Omron Sysmac Studio project Project-Backup-Onrom (Sysmac Studio 1.64.0.64008, StandardProject)

# Controller CLP: NX102-1020 version 1.33
Units and slaves: Unit 1 : NX-ID5442 (N1); Unit 2 : NX-OD5256 (N2); Unit 3 : NX-PF0730 (N3); Unit 5 : NX-SID800 (N5); Unit 6 : NX-SOD400 (N6)
Axis MC_Axis000, settings changed from default: AxisType=ServoType, UnitsConversion=EnumElement2, UnitsNumerator=8388608, UnitsDenominator=100, MaxVelocity=10000, MaxJogVelocity=8000, MaxAcceleration=50, MaxDeceleration=50, MaxPositiveTorqueLimit=050.0, MaxNegativeTorqueLimit=050.0, HomingMode=BackupAndProximitySignalOn, StartDirection=NegativeDirection, OriginInputDetectionDirection=NegativeDirection, HomingVelocity=100, HomingApproachVelocity=5, OriginCompensationValue=10, CompensationVelocity=5, ModuloMAXPosition=100, ModuloMINPosition=0, EncoderTypes=Abs
Task PrimaryTask (priority 4, period or condition 2000): Program0

VAR_GLOBAL
    PB1 : BOOL;  (* IHM; published *)
    O1 : BOOL;  (* at IOBus://unit#2/Output Bit 16 bits/Output Bit 01 *)
END_VAR
VAR_GLOBAL CONSTANT
    MC_Axis000 : _sAXIS_REF;  (* at MC://_MC_AX[0] *)
END_VAR
VAR_GLOBAL
    O2 : BOOL;  (* at IOBus://unit#2/Output Bit 16 bits/Output Bit 02 *)
    O3 : BOOL;  (* at IOBus://unit#2/Output Bit 16 bits/Output Bit 03 *)
    PBSET : BOOL;  (* IHM; published *)
    PBRESET : BOOL;  (* IHM; published *)
    PBMOMENT : BOOL;
    LPOUT02 : BOOL;
    LPOUT03 : BOOL;
    PBM_LIG : BOOL;  (* IHM; published *)
    PBM_DSL : BOOL;  (* IHM; published *)
    TEMPO_O2 : TIME;
    PV : DINT;
    SP : DINT;
    E001_Torque_actual_value : INT;  (* at ECAT://node#1/Torque actual value; published *)
    Torque_atual : INT;  (* IHM; published *)
END_VAR
VAR_GLOBAL RETAIN
    Set_torque : LREAL;  (* IHM; published *)
    Set_rampa : LREAL;  (* published *)
    Set_torque_veloc : LREAL;  (* IHM; published *)
    max_pos_torq : LREAL;  (* IHM; published *)
    max_neg_torq : LREAL;  (* IHM; published *)
END_VAR
VAR_GLOBAL
    E001_Position_actual_value : DINT;  (* at ECAT://node#1/Position actual value; published *)
    Pos_atual : DINT;  (* IHM; published *)
END_VAR
VAR_GLOBAL RETAIN
    Set_pos : LREAL;  (* IHM; published *)
    Set_veloc : LREAL;  (* IHM; published *)
END_VAR
VAR_GLOBAL
    READY_AXIS : BOOL;  (* IHM; published *)
    SERVO_ON : BOOL;  (* IHM; published *)
    Stop_servo : BOOL;  (* IHM; published *)
    RESET_ERRO : BOOL;  (* IHM; published *)
    RESET_OK : BOOL;  (* IHM; published *)
    TESET_TORQUE : BOOL;  (* IHM; published *)
    TORQUE_OK : BOOL;  (* IHM; published *)
    TORQUE_RUN : BOOL;  (* IHM; published *)
    sent_torque : BOOL;  (* IHM; published *)
    START_POS : BOOL;  (* IHM; published *)
    JOG_FWD : BOOL;  (* IHM; published *)
    JOG_REV : BOOL;  (* IHM; published *)
    JOG_AXIS1 : BOOL;  (* IHM; published *)
    JOG_AXIS2 : BOOL;  (* IHM; published *)
END_VAR
VAR_GLOBAL RETAIN
    Set_veloc_jog : LREAL;  (* IHM; published *)
END_VAR
VAR_GLOBAL
    E001_Minor_Fault : BOOL;  (* at ECAT://node#1/Sysmac Error Status/Minor Fault *)
    ERRO_OK : BOOL;  (* IHM; published *)
    E001_STO1 : BOOL;  (* STO Segurança; at ECAT://node#1/Digital inputs/STO1 *)
    mcAbsolute : _eMC_MOVE_MODE;
    mcRelative : _eMC_MOVE_MODE;
    mode_move : BOOL;
    selec_mode : _eMC_MOVE_MODE;
END_VAR
VAR_GLOBAL RETAIN
    START_POS_REL : BOOL;  (* published *)
    SET_POS_REL : LREAL;  (* published *)
    SET_VEL_REL : LREAL;  (* published *)
END_VAR
VAR_GLOBAL
    Emergencia_acionada_painel : BOOL;  (* published *)
    IHM_PL_EMERGENCIA : BOOL;  (* PL EMERGENCIA IHM *)
    TEMPO_REST_IHM : TIME;  (* Mostrar tempo IHM; published *)
    erro_servo : BOOL;  (* erro do servo *)
    ihm_PL_Barreira : BOOL;  (* Barreira IHM *)
    Emergencia_CLP : BOOL;  (* at IOBus://unit#5/Standard Input 1st Word/Si04 Logical Value *)
    PB_Reset_Seg_IHM : BOOL;  (* at IOBus://unit#4/Reset_IHM *)
    pb_reset_seg : BOOL;
    N5_Si01_Logical_Value : BOOL;  (* at IOBus://unit#5/Standard Input 1st Word/Si01 Logical Value; published *)
    N5_Si02_Logical_Value : BOOL;  (* at IOBus://unit#5/Standard Input 1st Word/Si02 Logical Value *)
    N6_So00_Status : BOOL;  (* at IOBus://unit#6/Standard Input 2nd Byte/So00 Status; published *)
    N6_So00_Monitor_Value : BOOL;  (* at IOBus://unit#6/Standard Input 1st Byte/So00 Monitor Value *)
END_VAR

(* Program Program0: safety or other program stored in binary form, left out *)

PROGRAM Program0
VAR
    PBSE : BOOL;
    AUX : BOOL;
    TON_O2 : TON;
    power_axis : MC_Power;
    jog_aixs : MC_MoveJog;
    move_axis : MC_Move;
    pos_axis : LREAL;
    pos_veloc : LREAL;
    Home_axis1 : MC_Home;
    reset1 : MC_Reset;
    torque_axis : MC_TorqueControl;
    limit_torque : MC_SetTorqueLimit;
    control1 : MC_TorqueControl;
    limit_torque_ok : BOOL;
    valor_torque : LREAL;
    timer_torque : LREAL;
    veloc_torque : LREAL;
    direction_torque : _eMC_DIRECTION;
    mode : _eMC_BUFFER_MODE;
    mode_stop : _eMC_BUFFER_MODE;
    mode_2 : _eMC_BUFFER_MODE;
    stop1 : MC_Stop;
    STOP_ON : BOOL;
    STOP_SET : BOOL;
    torque_pos : BOOL;
    torque_neg : BOOL;
    valor_torque_neg : LREAL;
    STOP_NEG : BOOL;
    BLOQUEAR : BOOL;
    mode3 : _eMC_BUFFER_MODE;
    HOME_1 : MC_Home;
    MOTOR1 : BOOL;
    Torque_pos_valor : LREAL;
    Torque_neg_valor : LREAL;
    MOVE_RELATIVE : MC_MoveRelative;
    Skt_TCP_ON : BOOL;
    Socket_TCP : _sSOCKET;
    SendDat_TCP : ARRAY[0..1999] OF BYTE;
    RcvDat_TCP : ARRAY[0..1999] OF BYTE;
    Connect_1 : SktTCPConnect;
    CleaBuf_1 : SktClearBuf;
    Status_1 : SktGetTCPStatus;
    RcvTCP : SktTCPRcv;
    CloseTCP : SktClose;
    Send_1 : SktTCPSend;
    linkTCP : BOOL;
    TCPCOM : BOOL;
    SENDOK : BOOL;
    Comun_open : BOOL;
    SendDatFH : STRING[255];
    SendDatSize : UINT;
    setDADOS : BOOL;
    ERRO_TCP1 : WORD;
    BusyRcv : BOOL;
    FHRcvDat : STRING[256];
    resutDat : UINT;
    resutData : DINT;
    veloc_JOG : LREAL;  (* Velocidade JOG *)
    veloc_REL : LREAL;  (* Velocidade Relativa *)
    veloc_Abs : LREAL;  (* Velocidade Absoluto *)
    Teste_SHL : LWORD;
    exemplo : BOOL;
END_VAR
VAR_EXTERNAL
    PB1 : BOOL;
    O1 : BOOL;
    PBSET : BOOL;
    O2 : BOOL;
    PBRESET : BOOL;
    PBMOMENT : BOOL;
    O3 : BOOL;
    LPOUT03 : BOOL;
    LPOUT02 : BOOL;
    PBM_LIG : BOOL;
    PBM_DSL : BOOL;
    TEMPO_O2 : TIME;
END_VAR
VAR_EXTERNAL CONSTANT
    MC_Axis000 : _sAXIS_REF;
END_VAR
VAR_EXTERNAL
    PV : DINT;
    SP : DINT;
    E001_Torque_actual_value : INT;
    E001_Position_actual_value : DINT;
    READY_AXIS : BOOL;
    SERVO_ON : BOOL;
    RESET_ERRO : BOOL;
    JOG_FWD : BOOL;
    JOG_REV : BOOL;
    JOG_AXIS2 : BOOL;
    JOG_AXIS1 : BOOL;
    START_POS : BOOL;
    RESET_OK : BOOL;
    TESET_TORQUE : BOOL;
    TORQUE_OK : BOOL;
    TORQUE_RUN : BOOL;
    Torque_atual : INT;
    Pos_atual : DINT;
    Set_pos : LREAL;
    Set_veloc : LREAL;
    Set_veloc_jog : LREAL;
    Set_torque : LREAL;
    Set_rampa : LREAL;
    Set_torque_veloc : LREAL;
    E001_Minor_Fault : BOOL;
    ERRO_OK : BOOL;
    max_pos_torq : LREAL;
    max_neg_torq : LREAL;
    sent_torque : BOOL;
    mcAbsolute : _eMC_MOVE_MODE;
    mcRelative : _eMC_MOVE_MODE;
    mode_move : BOOL;
    selec_mode : _eMC_MOVE_MODE;
    Stop_servo : BOOL;
    START_POS_REL : BOOL;
    SET_POS_REL : LREAL;
    SET_VEL_REL : LREAL;
END_VAR
VAR_EXTERNAL CONSTANT
    _EIP_EtnOnlineSta : BOOL;
END_VAR
VAR_EXTERNAL
    Emergencia_acionada_painel : BOOL;  (* Emergencia Acionada *)
    E001_STO1 : BOOL;
    IHM_PL_EMERGENCIA : BOOL;  (* PL EMERGENCIA IHM *)
    TEMPO_REST_IHM : TIME;  (* Mostrar tempo IHM *)
END_VAR
VAR_EXTERNAL CONSTANT
    _MC_AX : ARRAY[0..15] OF _sAXIS_REF;
END_VAR
VAR_EXTERNAL
    erro_servo : BOOL;  (* erro do servo *)
    ihm_PL_Barreira : BOOL;  (* Barreira IHM *)
    Emergencia_CLP : BOOL;  (* emergencia acionada no CLP de segurança *)
    PB_Reset_Seg_IHM : BOOL;  (* Reset da IHM para CLP Segurança *)
    pb_reset_seg : BOOL;  (* Reset Segurança *)
    N5_Si02_Logical_Value : BOOL;
    N6_So00_Status : BOOL;  (* Preparativo *)
    N6_So00_Monitor_Value : BOOL;  (* Preparativo *)
END_VAR
VAR
    _e1 : R_TRIG;
    _e2 : R_TRIG;
    _e3 : R_TRIG;
    _e4 : R_TRIG;
    _e5 : R_TRIG;
    _e6 : R_TRIG;
    _e7 : R_TRIG;
END_VAR

(* Section Section0: ladder, written here as Structured Text *)

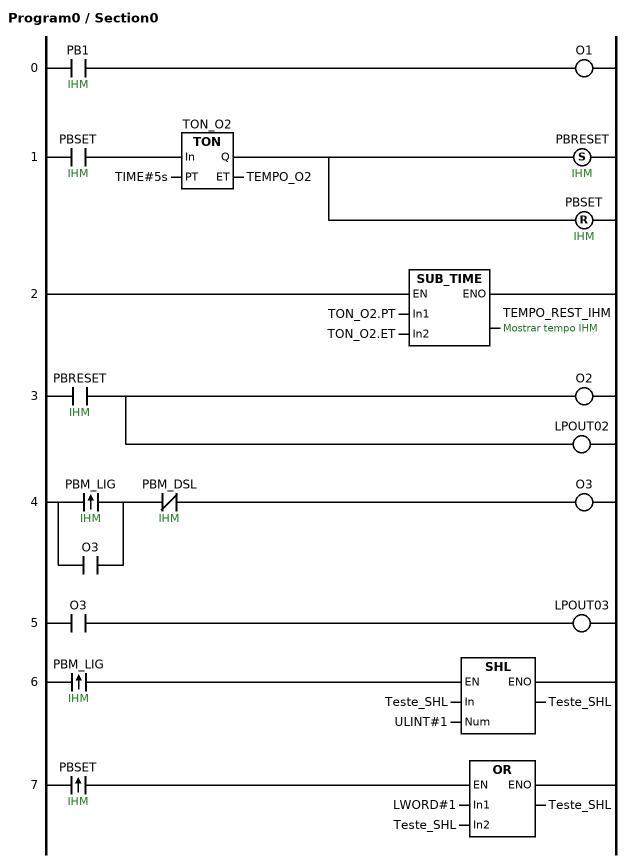
(* Rung 0 *)
O1 := PB1;
(* Rung 1 *)
TON_O2(In := PBSET, PT := TIME#5s, ET => TEMPO_O2);
IF TON_O2.Q THEN
    PBRESET := TRUE;
    PBSET := FALSE;
END_IF;
(* Rung 2 *)
TEMPO_REST_IHM := SUB_TIME(In1 := TON_O2.PT, In2 := TON_O2.ET);
(* Rung 3 *)
O2 := PBRESET;
LPOUT02 := PBRESET;
(* Rung 4 *)
_e1(CLK := PBM_LIG);
O3 := (_e1.Q OR O3) AND NOT PBM_DSL;
(* Rung 5 *)
LPOUT03 := O3;
(* Rung 6 *)
_e2(CLK := PBM_LIG);
IF _e2.Q THEN Teste_SHL := SHL(In := Teste_SHL, Num := ULINT#1); END_IF;
(* Rung 7 *)
_e3(CLK := PBSET);
IF _e3.Q THEN Teste_SHL := LWORD#1 OR Teste_SHL; END_IF;

(* Section Servo: ladder, written here as Structured Text *)

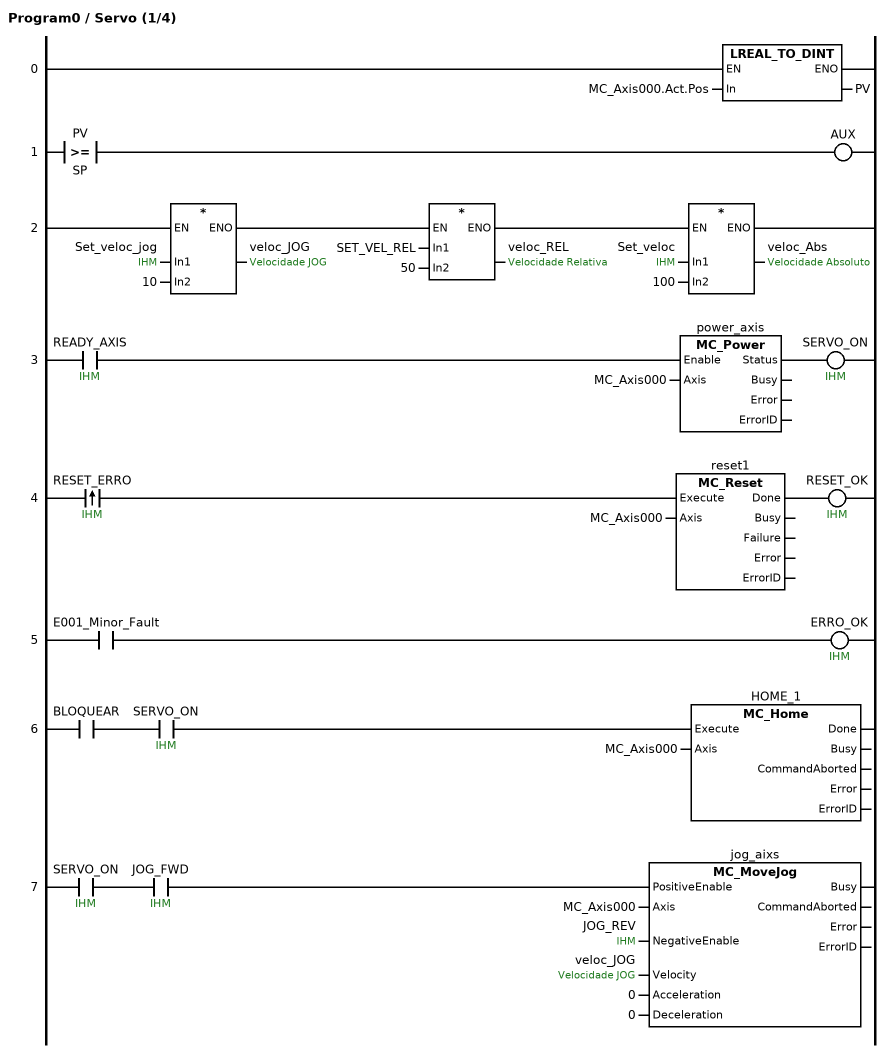
(* Rung 0 *)
PV := LREAL_TO_DINT(In := MC_Axis000.Act.Pos);
(* Rung 1 *)
AUX := PV >= SP;
(* Rung 2 *)
veloc_JOG := Set_veloc_jog * 10;
veloc_REL := SET_VEL_REL * 50;
veloc_Abs := Set_veloc * 100;
(* Rung 3 *)
power_axis(Enable := READY_AXIS, Axis := MC_Axis000);
SERVO_ON := power_axis.Status;
(* Rung 4 *)
_e4(CLK := RESET_ERRO);
reset1(Execute := _e4.Q, Axis := MC_Axis000);
RESET_OK := reset1.Done;
(* Rung 5 *)
ERRO_OK := E001_Minor_Fault;
(* Rung 6 *)
HOME_1(Execute := BLOQUEAR AND SERVO_ON, Axis := MC_Axis000);
(* Rung 7 *)
jog_aixs(PositiveEnable := SERVO_ON AND JOG_FWD, Axis := MC_Axis000, NegativeEnable := JOG_REV, Velocity := veloc_JOG, Acceleration := 0, Deceleration := 0);

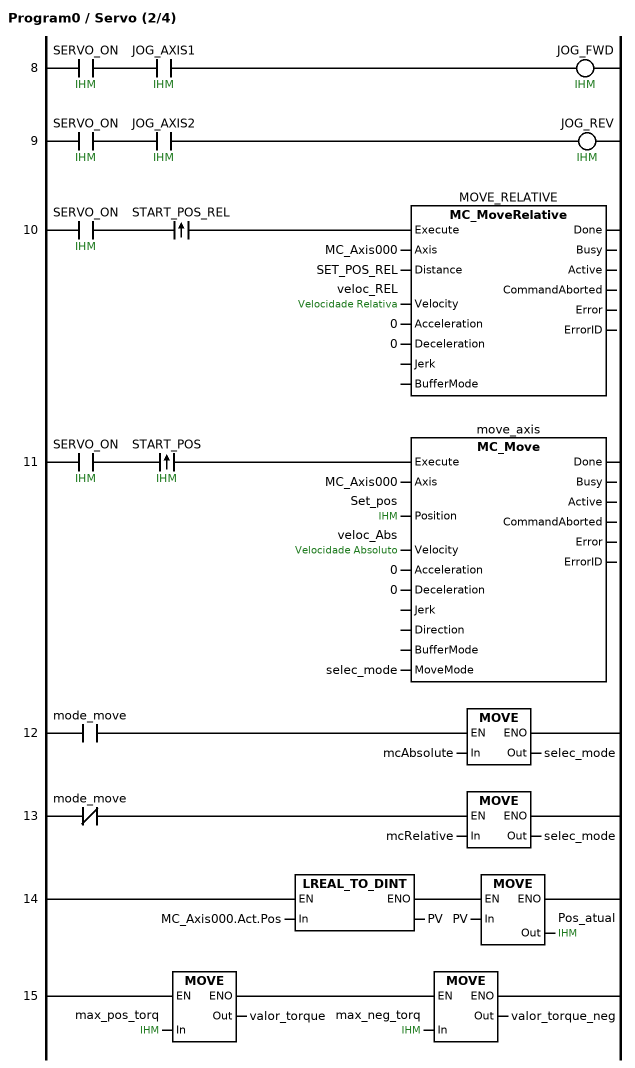
(* Rung 8 *)
JOG_FWD := SERVO_ON AND JOG_AXIS1;
(* Rung 9 *)
JOG_REV := SERVO_ON AND JOG_AXIS2;
(* Rung 10 *)
_e5(CLK := START_POS_REL);
MOVE_RELATIVE(Execute := SERVO_ON AND _e5.Q, Axis := MC_Axis000, Distance := SET_POS_REL, Velocity := veloc_REL, Acceleration := 0, Deceleration := 0);
(* Rung 11 *)
_e6(CLK := START_POS);
move_axis(Execute := SERVO_ON AND _e6.Q, Axis := MC_Axis000, Position := Set_pos, Velocity := veloc_Abs, Acceleration := 0, Deceleration := 0, MoveMode := selec_mode);
(* Rung 12 *)
IF mode_move THEN selec_mode := mcAbsolute; END_IF;
(* Rung 13 *)
IF NOT mode_move THEN selec_mode := mcRelative; END_IF;
(* Rung 14 *)
PV := LREAL_TO_DINT(In := MC_Axis000.Act.Pos);
Pos_atual := PV;
(* Rung 15 *)
valor_torque := max_pos_torq;
valor_torque_neg := max_neg_torq;

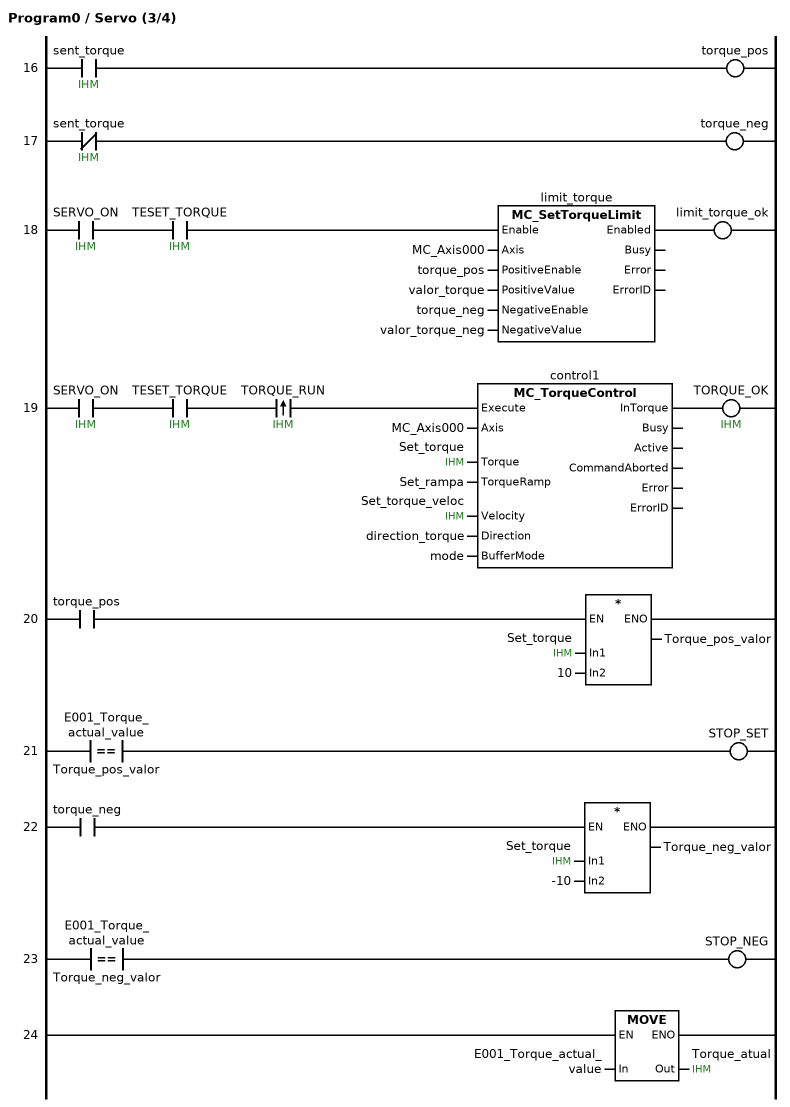
(* Rung 16 *)
torque_pos := sent_torque;
(* Rung 17 *)
torque_neg := NOT sent_torque;
(* Rung 18 *)
limit_torque(Enable := SERVO_ON AND TESET_TORQUE, Axis := MC_Axis000, PositiveEnable := torque_pos, PositiveValue := valor_torque, NegativeEnable := torque_neg, NegativeValue := valor_torque_neg);
limit_torque_ok := limit_torque.Enabled;
(* Rung 19 *)
_e7(CLK := TORQUE_RUN);
control1(Execute := SERVO_ON AND TESET_TORQUE AND _e7.Q, Axis := MC_Axis000, Torque := Set_torque, TorqueRamp := Set_rampa, Velocity := Set_torque_veloc, Direction := direction_torque, BufferMode := mode);
TORQUE_OK := control1.InTorque;
(* Rung 20 *)
IF torque_pos THEN Torque_pos_valor := Set_torque * 10; END_IF;
(* Rung 21 *)
STOP_SET := E001_Torque_actual_value = Torque_pos_valor;
(* Rung 22 *)
IF torque_neg THEN Torque_neg_valor := Set_torque * -10; END_IF;
(* Rung 23 *)
STOP_NEG := E001_Torque_actual_value = Torque_neg_valor;
(* Rung 24 *)
Torque_atual := E001_Torque_actual_value;

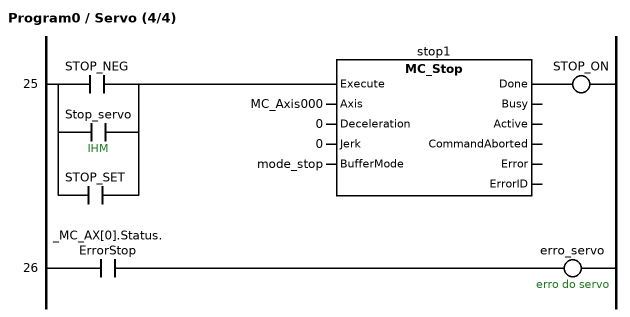
(* Rung 25 *)
stop1(Execute := STOP_NEG OR Stop_servo OR STOP_SET, Axis := MC_Axis000, Deceleration := 0, Jerk := 0, BufferMode := mode_stop);
STOP_ON := stop1.Done;
(* Rung 26 *)
erro_servo := _MC_AX[0].Status.ErrorStop;

(* Section TCP_Socket: ladder, written here as Structured Text *)

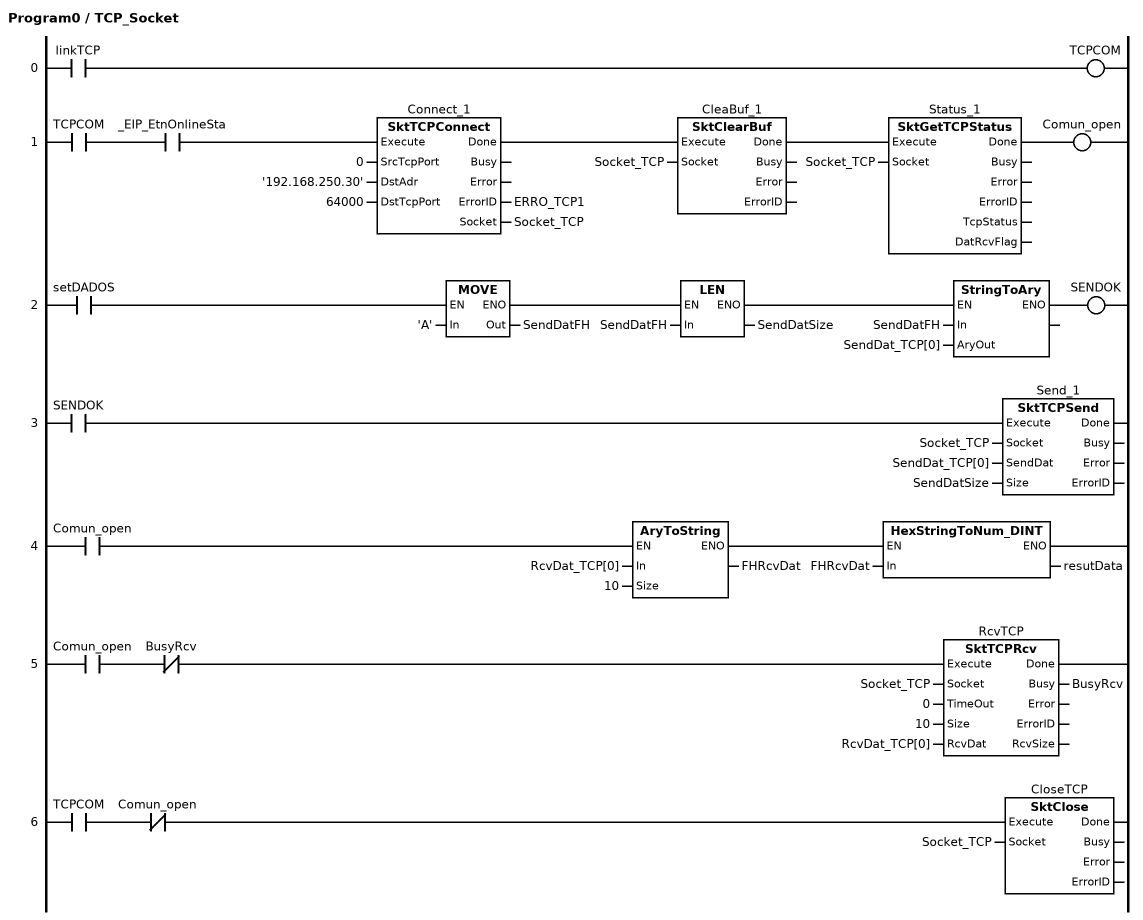
(* Rung 0 *)
TCPCOM := linkTCP;
(* Rung 1 *)
Connect_1(Execute := TCPCOM AND _EIP_EtnOnlineSta, SrcTcpPort := 0, DstAdr := '192.168.250.30', DstTcpPort := 64000, ErrorID => ERRO_TCP1, Socket => Socket_TCP);
CleaBuf_1(Execute := Connect_1.Done, Socket := Socket_TCP);
Status_1(Execute := CleaBuf_1.Done, Socket := Socket_TCP);
Comun_open := Status_1.Done;
(* Rung 2 *)
IF setDADOS THEN
    SendDatFH := 'A';
    SendDatSize := LEN(In := SendDatFH);
    StringToAry(In := SendDatFH, AryOut := SendDat_TCP[0]);
END_IF;
SENDOK := setDADOS;
(* Rung 3 *)
Send_1(Execute := SENDOK, Socket := Socket_TCP, SendDat := SendDat_TCP[0], Size := SendDatSize);
(* Rung 4 *)
IF Comun_open THEN
    FHRcvDat := AryToString(In := RcvDat_TCP[0], Size := 10);
    resutData := HexStringToNum_DINT(In := FHRcvDat);
END_IF;
(* Rung 5 *)
RcvTCP(Execute := Comun_open AND NOT BusyRcv, Socket := Socket_TCP, TimeOut := 0, Size := 10, RcvDat := RcvDat_TCP[0], Busy => BusyRcv);
(* Rung 6 *)
CloseTCP(Execute := TCPCOM AND NOT Comun_open, Socket := Socket_TCP);

(* Section Segurança: ladder, written here as Structured Text *)

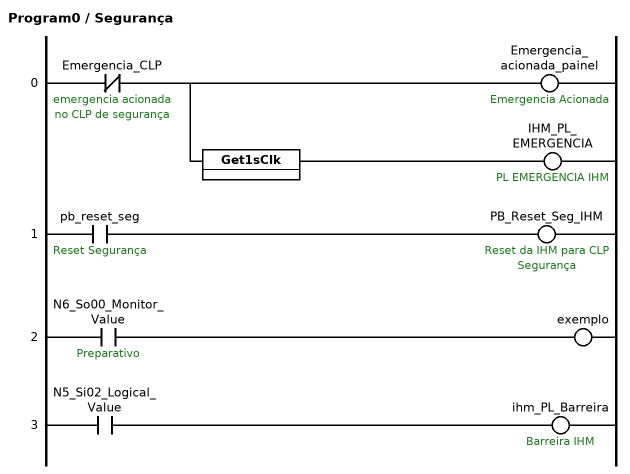
(* Rung 0 *)
Emergencia_acionada_painel := NOT Emergencia_CLP;
IHM_PL_EMERGENCIA := NOT Emergencia_CLP AND Get1sClk();
(* Rung 1 *)
PB_Reset_Seg_IHM := pb_reset_seg;
(* Rung 2 *)
exemplo := N6_So00_Monitor_Value;
(* Rung 3 *)
ihm_PL_Barreira := N5_Si02_Logical_Value;
END_PROGRAM

# Device HMI (NA): not converted